# EPICS IOC start-up script: iocsh/evmi.iocsh
# .init.iocsh
# ===========

mrmEvgSetupPCI($(DEV), $(PCIID))

dbLoadRecords("evm-mtca-300-ess.db", "SYS=$(IOC), D=$(DEV), EVG=$(DEV), FEVT=$(TS_CLK), FRF=$(TS_CLK), RFDIV=1")

var evrMrmTimeNSOverflowThreshold 1000000

#EOF
